// TIA Portal V17 export
// export: Created 2023-03-06T02:05:27.3380999Z, ExportSetting WithDefaults, DisplayName Totally Integrated Automation Portal, DisplayVersion V17 Update 4, DisplayName TIA Portal Openness, DisplayVersion V17 Update 4, DisplayName TIA Portal Version Control Interface, DisplayVersion V17, DisplayName STEP 7 Professional, DisplayVersion V17 Update 4, DisplayName STEP 7 Safety, DisplayVersion V17, DisplayName WinCC Professional, DisplayVersion V17 Update 4
TYPE "W_MV"
// stored: IsFailsafeCompliant false
   STRUCT
      xCircBrk1OpenCmd : Bool;   // U13.DI0.4
      xCircBrk1CloseCmd : Bool;   // U13.DI0.5
      xLVCircBrk1OpenCmd : Bool;   // U13.DI0.4
      xLVCircBrk1CloseCmd : Bool;   // U13.DI0.5
      xCircBrk2OpenCmd : Bool;   // U13.DI0.4
      xCircBrk2CloseCmd : Bool;   // U13.DI0.5
      xLVCircBrk2OpenCmd : Bool;   // U13.DI0.4
      xLVCircBrk2CloseCmd : Bool;   // U13.DI0.5
   END_STRUCT;
END_TYPE
